{attribute addProperty BoxType "EK1100-0000-0018"}
{attribute addProperty Id "Beckhoff_EL9xxxEK1122Beckhoff_EL9xxxEK1122_2D49AF05162A_0003_EL9110_0000_0016EL9110_AE5731BA263.25A_0004_EL9110_0000_0017EL9110_AE5731BA263.25A_0005_EL9110_0000_0018EL9110_AE5731BA263.25A_0006_EL9160_0000_0016EL9160_AE5731BA263.25A_0007_EL9210_0000_0016EL9210_B219644D344.25A_0008_EL9210_0000_0017EL9210_B219644D344.25A_0009_EL9210_0000_0018EL9210_B219644D344.25A_0010_EL9210_0020_0016EL9210_B219644D344.25A_0011_EL9210_0020_0017EL9210_B219644D344.25A_0012_EL9210_0020_0018EL9210_B219644D344.25A_0013_EL9221_4030_0018EL9221_E4BC007313016.25A_0014_EL9221_5000_0018EL9221_E4BC007313016.25A_0015_EL9221_5090_0018EL9221_E4BC007313016.25A_0016_EL9221_6000_0018EL9221_E4BC007313016.25A_0017_EL9221_6040_0018EL9221_E4BC007313016.25A_0018_EL9221_9060_0018EL9221_E4BC007313016.25A_0019_EL9221_9080_0018EL9221_E4BC007313016.25A_0020_EL9222_4433_0018EL9222_5848358917822.25A_0021_EL9222_5500_0018EL9222_5848358917822.25A_0022_EL9222_6600_0018EL9222_5848358917822.25A_0023_EL9222_6644_0018EL9222_5848358917822.25A_0024_EL9222_9482_0018EL9222_5848358917822.25A_0025_EL9222_9664_0018EL9222_5848358917822.25A_0026_EL9227_4433_0018EL9227_9D6FA8BB30638.25A_0027_EL9227_5500_0018EL9227_9D6FA8BB30638.25A_0028_EL9227_6600_0018EL9227_9D6FA8BB30638.25A_0029_EL9227_6644_0018EL9227_9D6FA8BB30638.25A_0030_EL9227_9482_0018EL9227_9D6FA8BB30638.25A_0031_EL9227_9664_0018EL9227_9D6FA8BB30638.25A_0032_EL9260_0000_0016EL9260_B219644D344.25A_0033_EL9410_0000_0016EL9410_0EEAC8F2344.25A_0034_EL9410_0000_0017EL9410_0EEAC8F2344.25A_0035_EL9505_0000_0016EL9505_13AAEB7E344.25A_0036_EL9505_0000_0017EL9505_13AAEB7E344.25A_0037_EL9505_0000_0018EL9505_13AAEB7E344.25A_0038_EL9508_0000_0016EL9508_13AAEB7E344.25A_0039_EL9508_0000_0017EL9508_13AAEB7E344.25A_0040_EL9508_0000_0018EL9508_13AAEB7E344.25A_0041_EL9510_0000_0016EL9510_13AAEB7E344.25A_0042_EL9510_0000_0017EL9510_13AAEB7E344.25A_0043_EL9510_0000_0018EL9510_13AAEB7E344.25A_0044_EL9512_0000_0016EL9512_13AAEB7E344.25A_0045_EL9512_0000_0017EL9512_13AAEB7E344.25A_0046_EL9512_0000_0018EL9512_13AAEB7E344.25A_0047_EL9515_0000_0016EL9515_13AAEB7E344.25A_0048_EL9515_0000_0017EL9515_13AAEB7E344.25A_0049_EL9515_0000_0018EL9515_13AAEB7E344.25A_0050_EL9520_0000_0016EL9520_B21A9EBB263.25A_0051_EL9520_0000_0017EL9520_B21A9EBB263.25A_0052_EL9540_0010_0016EL9540_081B367B344.25A_0053_EL9550_0010_0016EL9550_B50CDD11506.25A_0054_EL9560_0000_0016EL9560_84A42FC9344.25A_0055_EL9560_0000_0017EL9560_84A42FC9344.25A_0056_EL9560_0000_0018EL9560_84A42FC9344.25A_0057_EL9576_0000_0016EL9576_06679F7620225.25A_0058_EL9576_0000_0017EL9576_30D5723B21026.25A_0059_EL9576_0000_0018EL9576_30D5723B21026.25A_0060_EL9576_0000_0019EL9576_8602C5C421827.25A_0061_EL9576_0000_0020EL9576_EB67CEB421026.25A_0062_EL9576_0000_0021EL9576_EB67CEB421026.25A_0063_EL9576_0000_0022EL9576_EEF1625221827.25A_0086_EL9540_0010EL9540_081B367B344.25A_0088_EL9550_0010EL9550_B50CDD11506.25"}
{attribute addProperty CRC "2217289967"}
{attribute addProperty SizeInBites "6550"}
{attribute addProperty SizeInBytes "818.75"}
TYPE Beckhoff_EL9xxx_842928EF EXTENDS EK1100_179A0949 :
STRUCT
	{attribute addProperty Name "Beckhoff_EL9xxxEK1122"}
	Beckhoff_EL9xxxEK1122 : Beckhoff_EL9xxxEK1122_2D49AF05;
	{attribute addProperty Name "A_0003_EL9110_0000_0016"}
	A_0003_EL9110_0000_0016 : EL9110_AE5731BA;
	{attribute addProperty Name "A_0004_EL9110_0000_0017"}
	A_0004_EL9110_0000_0017 : EL9110_AE5731BA;
	{attribute addProperty Name "A_0005_EL9110_0000_0018"}
	A_0005_EL9110_0000_0018 : EL9110_AE5731BA;
	{attribute addProperty Name "A_0006_EL9160_0000_0016"}
	A_0006_EL9160_0000_0016 : EL9160_AE5731BA;
	{attribute addProperty Name "A_0007_EL9210_0000_0016"}
	A_0007_EL9210_0000_0016 : EL9210_B219644D;
	{attribute addProperty Name "A_0008_EL9210_0000_0017"}
	A_0008_EL9210_0000_0017 : EL9210_B219644D;
	{attribute addProperty Name "A_0009_EL9210_0000_0018"}
	A_0009_EL9210_0000_0018 : EL9210_B219644D;
	{attribute addProperty Name "A_0010_EL9210_0020_0016"}
	A_0010_EL9210_0020_0016 : EL9210_B219644D;
	{attribute addProperty Name "A_0011_EL9210_0020_0017"}
	A_0011_EL9210_0020_0017 : EL9210_B219644D;
	{attribute addProperty Name "A_0012_EL9210_0020_0018"}
	A_0012_EL9210_0020_0018 : EL9210_B219644D;
	{attribute addProperty Name "A_0013_EL9221_4030_0018"}
	A_0013_EL9221_4030_0018 : EL9221_E4BC0073;
	{attribute addProperty Name "A_0014_EL9221_5000_0018"}
	A_0014_EL9221_5000_0018 : EL9221_E4BC0073;
	{attribute addProperty Name "A_0015_EL9221_5090_0018"}
	A_0015_EL9221_5090_0018 : EL9221_E4BC0073;
	{attribute addProperty Name "A_0016_EL9221_6000_0018"}
	A_0016_EL9221_6000_0018 : EL9221_E4BC0073;
	{attribute addProperty Name "A_0017_EL9221_6040_0018"}
	A_0017_EL9221_6040_0018 : EL9221_E4BC0073;
	{attribute addProperty Name "A_0018_EL9221_9060_0018"}
	A_0018_EL9221_9060_0018 : EL9221_E4BC0073;
	{attribute addProperty Name "A_0019_EL9221_9080_0018"}
	A_0019_EL9221_9080_0018 : EL9221_E4BC0073;
	{attribute addProperty Name "A_0020_EL9222_4433_0018"}
	A_0020_EL9222_4433_0018 : EL9222_58483589;
	{attribute addProperty Name "A_0021_EL9222_5500_0018"}
	A_0021_EL9222_5500_0018 : EL9222_58483589;
	{attribute addProperty Name "A_0022_EL9222_6600_0018"}
	A_0022_EL9222_6600_0018 : EL9222_58483589;
	{attribute addProperty Name "A_0023_EL9222_6644_0018"}
	A_0023_EL9222_6644_0018 : EL9222_58483589;
	{attribute addProperty Name "A_0024_EL9222_9482_0018"}
	A_0024_EL9222_9482_0018 : EL9222_58483589;
	{attribute addProperty Name "A_0025_EL9222_9664_0018"}
	A_0025_EL9222_9664_0018 : EL9222_58483589;
	{attribute addProperty Name "A_0026_EL9227_4433_0018"}
	A_0026_EL9227_4433_0018 : EL9227_9D6FA8BB;
	{attribute addProperty Name "A_0027_EL9227_5500_0018"}
	A_0027_EL9227_5500_0018 : EL9227_9D6FA8BB;
	{attribute addProperty Name "A_0028_EL9227_6600_0018"}
	A_0028_EL9227_6600_0018 : EL9227_9D6FA8BB;
	{attribute addProperty Name "A_0029_EL9227_6644_0018"}
	A_0029_EL9227_6644_0018 : EL9227_9D6FA8BB;
	{attribute addProperty Name "A_0030_EL9227_9482_0018"}
	A_0030_EL9227_9482_0018 : EL9227_9D6FA8BB;
	{attribute addProperty Name "A_0031_EL9227_9664_0018"}
	A_0031_EL9227_9664_0018 : EL9227_9D6FA8BB;
	{attribute addProperty Name "A_0032_EL9260_0000_0016"}
	A_0032_EL9260_0000_0016 : EL9260_B219644D;
	{attribute addProperty Name "A_0033_EL9410_0000_0016"}
	A_0033_EL9410_0000_0016 : EL9410_0EEAC8F2;
	{attribute addProperty Name "A_0034_EL9410_0000_0017"}
	A_0034_EL9410_0000_0017 : EL9410_0EEAC8F2;
	{attribute addProperty Name "A_0035_EL9505_0000_0016"}
	A_0035_EL9505_0000_0016 : EL9505_13AAEB7E;
	{attribute addProperty Name "A_0036_EL9505_0000_0017"}
	A_0036_EL9505_0000_0017 : EL9505_13AAEB7E;
	{attribute addProperty Name "A_0037_EL9505_0000_0018"}
	A_0037_EL9505_0000_0018 : EL9505_13AAEB7E;
	{attribute addProperty Name "A_0038_EL9508_0000_0016"}
	A_0038_EL9508_0000_0016 : EL9508_13AAEB7E;
	{attribute addProperty Name "A_0039_EL9508_0000_0017"}
	A_0039_EL9508_0000_0017 : EL9508_13AAEB7E;
	{attribute addProperty Name "A_0040_EL9508_0000_0018"}
	A_0040_EL9508_0000_0018 : EL9508_13AAEB7E;
	{attribute addProperty Name "A_0041_EL9510_0000_0016"}
	A_0041_EL9510_0000_0016 : EL9510_13AAEB7E;
	{attribute addProperty Name "A_0042_EL9510_0000_0017"}
	A_0042_EL9510_0000_0017 : EL9510_13AAEB7E;
	{attribute addProperty Name "A_0043_EL9510_0000_0018"}
	A_0043_EL9510_0000_0018 : EL9510_13AAEB7E;
	{attribute addProperty Name "A_0044_EL9512_0000_0016"}
	A_0044_EL9512_0000_0016 : EL9512_13AAEB7E;
	{attribute addProperty Name "A_0045_EL9512_0000_0017"}
	A_0045_EL9512_0000_0017 : EL9512_13AAEB7E;
	{attribute addProperty Name "A_0046_EL9512_0000_0018"}
	A_0046_EL9512_0000_0018 : EL9512_13AAEB7E;
	{attribute addProperty Name "A_0047_EL9515_0000_0016"}
	A_0047_EL9515_0000_0016 : EL9515_13AAEB7E;
	{attribute addProperty Name "A_0048_EL9515_0000_0017"}
	A_0048_EL9515_0000_0017 : EL9515_13AAEB7E;
	{attribute addProperty Name "A_0049_EL9515_0000_0018"}
	A_0049_EL9515_0000_0018 : EL9515_13AAEB7E;
	{attribute addProperty Name "A_0050_EL9520_0000_0016"}
	A_0050_EL9520_0000_0016 : EL9520_B21A9EBB;
	{attribute addProperty Name "A_0051_EL9520_0000_0017"}
	A_0051_EL9520_0000_0017 : EL9520_B21A9EBB;
	{attribute addProperty Name "A_0052_EL9540_0010_0016"}
	A_0052_EL9540_0010_0016 : EL9540_081B367B;
	{attribute addProperty Name "A_0053_EL9550_0010_0016"}
	A_0053_EL9550_0010_0016 : EL9550_B50CDD11;
	{attribute addProperty Name "A_0054_EL9560_0000_0016"}
	A_0054_EL9560_0000_0016 : EL9560_84A42FC9;
	{attribute addProperty Name "A_0055_EL9560_0000_0017"}
	A_0055_EL9560_0000_0017 : EL9560_84A42FC9;
	{attribute addProperty Name "A_0056_EL9560_0000_0018"}
	A_0056_EL9560_0000_0018 : EL9560_84A42FC9;
	{attribute addProperty Name "A_0057_EL9576_0000_0016"}
	A_0057_EL9576_0000_0016 : EL9576_06679F76;
	{attribute addProperty Name "A_0058_EL9576_0000_0017"}
	A_0058_EL9576_0000_0017 : EL9576_30D5723B;
	{attribute addProperty Name "A_0059_EL9576_0000_0018"}
	A_0059_EL9576_0000_0018 : EL9576_30D5723B;
	{attribute addProperty Name "A_0060_EL9576_0000_0019"}
	A_0060_EL9576_0000_0019 : EL9576_8602C5C4;
	{attribute addProperty Name "A_0061_EL9576_0000_0020"}
	A_0061_EL9576_0000_0020 : EL9576_EB67CEB4;
	{attribute addProperty Name "A_0062_EL9576_0000_0021"}
	A_0062_EL9576_0000_0021 : EL9576_EB67CEB4;
	{attribute addProperty Name "A_0063_EL9576_0000_0022"}
	A_0063_EL9576_0000_0022 : EL9576_EEF16252;
	{attribute addProperty Name "A_0086_EL9540_0010"}
	A_0086_EL9540_0010 : EL9540_081B367B;
	{attribute addProperty Name "A_0088_EL9550_0010"}
	A_0088_EL9550_0010 : EL9550_B50CDD11;
END_STRUCT
END_TYPE

(* stored: Version 1.2.0.0, ProductVersion 3.1.4024.9
   DUT Beckhoff_EL9xxx_842928EF: Id {db12182d-8a3f-4572-883f-13da381bc842} *)
